// TwinCAT 3 PLC project Desktop
// ProgramVersion: 3.1.4020.1
// CompilerDefines: VISU_USEWSTRING
// libraries:
//   Standard, * (System)
//   VisuElems, 3.5.6.10 (System)
//   VisuElemsSpecialControls, 3.5.6.0 (System)
//   VisuElemsWinControls, 3.5.6.0 (System)
//   VisuElemTextEditor, 3.5.6.0 (System)
//   visuinputs, 3.5.6.0 (system)
//   VisuNativeControl, 3.5.6.0 (System)
//   Tc2_Math, * (Beckhoff Automation GmbH)
//   Tc2_MC2, * (Beckhoff Automation GmbH)
//   Tc2_NCI, * (Beckhoff Automation GmbH)
//   Tc2_NcKinematicTransformation, * (Beckhoff Automation GmbH)
//   Tc2_SPA, * (Beckhoff Automation GmbH)
//   Tc2_Standard, * (Beckhoff Automation GmbH)
//   Tc2_System, * (Beckhoff Automation GmbH)
//   Tc3_Interfaces, * (Beckhoff Automation GmbH)
//   Tc3_Module, * (Beckhoff Automation GmbH)
//   VisuDialogs, * (System)
// project tree:
//   / GlobalTextList.TcGTLO, PlcTask.TcTTO, Visualization Manager.TcVMO (not stored)
//   GVLs/ AxesCharacters.TcGVL, Functions.TcGVL, HardwareCharacters.TcGVL, ItpCharacters.TcGVL, KinCharacters.TcGVL
//   POUs/ Axes_Itp.TcPOU, Coordinate_System.TcPOU, Kinematics.TcPOU, Axes.TcPOU, Collision_Detection.TcPOU, MAIN.TcPOU, Home.TcPOU, Singularity.TcPOU, SoftFloat.TcPOU, UserFrames.TcPOU
//   VISUs/ CtrlPANEL.TcVIS, Home.TcVIS
// real-time tasks:
//   TASK PlcTask: cycle T#1ms, priority 1, ADS port 350
//   TASK VISU_TASK: cycle T#100000us, priority 10, ADS port 351
// motion (NC):
//   TASK NC-Task 1 SAF: cycle T#2ms, priority 4, ADS port 501
//   TASK NC-Task 1 SVB: cycle T#10ms, priority 8, ADS port 511
//   AXIS ACS M1 (id 1)
//     General: UnitName=Degree, UnitFlags=#x00000004
//     Dynamic: Acceleration=16333.3, Deceleration=16333.3, Jerk=111157
//     Velo: SlowManual=10, FastManual=20, Maximum=2500
//     OtherSettings: AllowMotionCmdToSlave=true
//     encoder EncType=1
//       EncPara: ScaleFactorNumerator=360, ScaleFactorDenominator=10485760, Offset=-437.0522
//         SoftEndMinControl: Enable=true, Range=-60
//         SoftEndMaxControl: Enable=true, Range=80
//     drive DrvType=5
//       Analog: VeloReferenz=2700
//       TimeComp: TaskDelayCycles=1
//     controller CtrType=1
//       CtrPara: PriorControlFactor=1
//         PID: PosKp=50
//         Observer: BandWidth=20
//   AXIS ACS M2 (id 2)
//     General: UnitName=Degree
//     Dynamic: Acceleration=16416.7, Deceleration=16416.7, Jerk=111137
//     Velo: SlowManual=10, FastManual=20, Maximum=2500
//     OtherSettings: AllowMotionCmdToSlave=true
//     encoder EncType=1
//       EncPara: ScaleFactorNumerator=360, ScaleFactorDenominator=10485760, Offset=-175.265
//         SoftEndMinControl: Enable=true, Range=-60
//         SoftEndMaxControl: Enable=true, Range=80
//     drive DrvType=5
//       Analog: VeloReferenz=2700
//       TimeComp: TaskDelayCycles=1
//     controller CtrType=1
//       CtrPara: PriorControlFactor=1
//         PID: PosKp=50
//         Observer: BandWidth=20
//   AXIS ACS M3 (id 3)
//     General: UnitName=Degree
//     Dynamic: Acceleration=16333.3, Deceleration=16333.3, Jerk=111157
//     Velo: SlowManual=10, FastManual=20, Maximum=2500
//     OtherSettings: AllowMotionCmdToSlave=true
//     encoder EncType=1
//       EncPara: ScaleFactorNumerator=360, ScaleFactorDenominator=10485760, Offset=-483.9976
//         SoftEndMinControl: Enable=true, Range=-60
//         SoftEndMaxControl: Enable=true, Range=80
//     drive DrvType=5
//       Analog: VeloReferenz=2700
//       TimeComp: TaskDelayCycles=1
//     controller CtrType=1
//       CtrPara: PriorControlFactor=1
//         PID: PosKp=50
//         Observer: BandWidth=20
//   AXIS MCS X (id 4)
//     Dynamic: Acceleration=16500, Deceleration=16500, Jerk=111122
//     Velo: SlowManual=50, FastManual=100, Maximum=2500
//     OtherSettings: AllowMotionCmdToSlave=true, PulseDistancePos=1, PulseDistanceNeg=1
//     encoder EncType=1
//       SoftEndMinControl: Range=-250
//       SoftEndMaxControl: Range=250
//     drive DrvType=5
//       Analog: VeloReferenz=3250
//       TimeComp: TaskDelayCycles=1
//     controller CtrType=1
//       CtrPara: PriorControlFactor=1
//         PID: PosKp=20
//         Observer: BandWidth=20
//   AXIS MCS Y (id 5)
//     Dynamic: Acceleration=16500, Deceleration=16500, Jerk=111122
//     Velo: SlowManual=50, FastManual=100, Maximum=2500
//     OtherSettings: AllowMotionCmdToSlave=true, PulseDistancePos=1, PulseDistanceNeg=1
//     encoder EncType=1
//       SoftEndMinControl: Range=-250
//       SoftEndMaxControl: Range=250
//     drive DrvType=5
//       Analog: VeloReferenz=3250
//       TimeComp: TaskDelayCycles=1
//     controller CtrType=1
//       CtrPara: PriorControlFactor=1
//         PID: PosKp=20
//         Observer: BandWidth=20
//   AXIS MCS Z (id 6)
//     Dynamic: Acceleration=16416.7, Deceleration=16416.7, Jerk=111137
//     Velo: SlowManual=50, FastManual=100, Maximum=2500
//     OtherSettings: AllowMotionCmdToSlave=true, PulseDistancePos=1, PulseDistanceNeg=1
//     encoder EncType=1
//       SoftEndMinControl: Range=-250
//       SoftEndMaxControl: Range=250
//     drive DrvType=5
//       Analog: VeloReferenz=3250
//       TimeComp: TaskDelayCycles=1
//     controller CtrType=1
//       CtrPara: PriorControlFactor=1
//         PID: PosKp=20
//         Observer: BandWidth=20
// variable links:
//   Desktop/Desktop Instance <-> NC-Task 1 SAF/Axes/ACS M1
//     PlcTask Inputs/AxesCharacters.MachX.NcToPlc <-> Outputs/ToPlc
//     PlcTask Outputs/AxesCharacters.MachX.PlcToNc <-> Inputs/FromPlc
//   Desktop/Desktop Instance <-> NC-Task 1 SAF/Axes/ACS M2
//     PlcTask Inputs/AxesCharacters.MachY.NcToPlc <-> Outputs/ToPlc
//     PlcTask Outputs/AxesCharacters.MachY.PlcToNc <-> Inputs/FromPlc
//   Desktop/Desktop Instance <-> NC-Task 1 SAF/Axes/ACS M3
//     PlcTask Inputs/AxesCharacters.MachZ.NcToPlc <-> Outputs/ToPlc
//     PlcTask Outputs/AxesCharacters.MachZ.PlcToNc <-> Inputs/FromPlc
//   Desktop/Desktop Instance <-> NC-Task 1 SAF/Axes/MCS X
//     PlcTask Inputs/AxesCharacters.SimsX.NcToPlc <-> Outputs/ToPlc
//     PlcTask Outputs/AxesCharacters.SimsX.PlcToNc <-> Inputs/FromPlc
//   Desktop/Desktop Instance <-> NC-Task 1 SAF/Axes/MCS Y
//     PlcTask Inputs/AxesCharacters.SimsY.NcToPlc <-> Outputs/ToPlc
//     PlcTask Outputs/AxesCharacters.SimsY.PlcToNc <-> Inputs/FromPlc
//   Desktop/Desktop Instance <-> NC-Task 1 SAF/Axes/MCS Z
//     PlcTask Inputs/AxesCharacters.SimsZ.NcToPlc <-> Outputs/ToPlc
//     PlcTask Outputs/AxesCharacters.SimsZ.PlcToNc <-> Inputs/FromPlc
//   Desktop/Desktop Instance <-> NC-Task 1 SAF/Kinametic_Channel
//     PlcTask Inputs/KinCharacters.in_stKinToPlc <-> Outputs/ToPlc
//     PlcTask Outputs/KinCharacters.out_stPlcTokin <-> Inputs/FromPlc
//   Desktop/Desktop Instance <-> NC-Task 1 SAF/NCI Interpolation
//     PlcTask Inputs/ItpCharacters.in_stItpToPLC <-> Outputs/ToPlc
//     PlcTask Outputs/ItpCharacters.out_stPLCToItp <-> Inputs/FromPlc

CONFIGURATION Desktop
    RESOURCE PLC ON TwinCAT3
        TASK PlcTask(INTERVAL := T#1ms, PRIORITY := 1);
        PROGRAM MAIN WITH PlcTask : MAIN;
    END_RESOURCE
END_CONFIGURATION

// ---- GVLs/AxesCharacters.TcGVL
VAR_GLOBAL
    in_uiMasterAxes_Override: LREAL := 100;
	in_bMasterAxes_Enable: BOOL ;    

    MachX: AXIS_REF;	
    in_bMachX_Enable: BOOL;
	in_uiMachX_Override: LREAL;
	out_bMachX_Status: BOOL;
	out_uiMachX_ErrorID: UDINT;
	
    MachY: AXIS_REF;
	in_bMachY_Enable: BOOL ;
	in_uiMachY_Override: LREAL;
	out_bMachY_Status: BOOL;
	out_uiMachY_ErrorID: UDINT;
	
    MachZ: AXIS_REF;
	in_bMachZ_Enable: BOOL ;
	in_uiMachZ_Override: LREAL;
	out_bMachZ_Status: BOOL;
	out_uiMachZ_ErrorID: UDINT;
	
    SimsX: AXIS_REF;
	in_bSimsX_Enable: BOOL ;
	in_uiSimsX_Override: LREAL;
	out_bSimsX_Status: BOOL;
	out_uiSimsX_ErrorID: UDINT;
	
    SimsY: AXIS_REF;
	in_bSimsY_Enable: BOOL ;
	in_uiSimsY_Override: LREAL;
	out_bSimsY_Status: BOOL;
	out_uiSimsY_ErrorID: UDINT;
	
    SimsZ: AXIS_REF;
	in_bSimsZ_Enable: BOOL ;
	in_uiSimsZ_Override: LREAL;
	out_bSimsZ_Status: BOOL;
	out_uiSimsZ_ErrorID: UDINT;
		
	in_bAxes_MachX_Jog_Forward: BOOL;
	in_bAxes_MachX_Jog_Backward: BOOL;
	out_uiAxes_MachX_Jog_ErrorID: UDINT;
		
	in_bAxes_MachY_Jog_Forward: BOOL;
	in_bAxes_MachY_Jog_Backward: BOOL;
	out_uiAxes_MachY_Jog_ErrorID: UDINT;
	
	in_bAxes_MachZ_Jog_Forward: BOOL;
	in_bAxes_MachZ_Jog_Backward: BOOL;
	out_uiAxes_MachZ_Jog_ErrorID: UDINT;
	
    in_bAxes_SimsX_Jog_Forward: BOOL;
	in_bAxes_SimsX_Jog_Backward: BOOL;
	out_uiAxes_SimsX_Jog_ErrorID: UDINT;
	
    in_bAxes_SimsY_Jog_Forward: BOOL;
	in_bAxes_SimsY_Jog_Backward: BOOL;
	out_uiAxes_SimsY_Jog_ErrorID: UDINT;
	
    in_bAxes_SimsZ_Jog_Forward: BOOL;
	in_bAxes_SimsZ_Jog_Backward: BOOL;
	out_uiAxes_SimsZ_Jog_ErrorID: UDINT;

	out_uiMachX_Error: BOOL;
	out_uiMachY_Error: BOOL;
	out_uiMachZ_Error: BOOL;
	out_uiSimsX_Error: BOOL;
	out_uiSimsY_Error: BOOL;
	out_uiSimsZ_Error: BOOL;
	out_bAxes_Master_Error: BOOL;
	
	Axes_Reset_All: BOOL;
		
END_VAR

// ---- GVLs/Functions.TcGVL
VAR_GLOBAL
	
// Move to Home Function
	in_b_MoveHome: BOOL;
	SimsX_Home_Done: BOOL;
	SimsY_Home_Done: BOOL;
	SimsZ_Home_Done: BOOL;
	
	Set_Pos_XHome: LREAL;
	Set_Pos_YHome: LREAL;
	Set_Pos_ZHome: LREAL;
	Set_Home_Override: LREAL:= 1000;
	out_b_inHome: BOOL;
	
END_VAR

// ---- GVLs/HardwareCharacters.TcGVL
VAR_GLOBAL
	in_bMasterAxes_Enable_HW AT %I*: BOOL;
	out_bMasterAxes_Enable_HW AT %Q*: BOOL;
	out_bSimsX_Axes_busy_HW AT %Q*: BOOL;
	out_bSimsY_Axes_busy_HW AT %Q*: BOOL;
	out_bSimsZ_Axes_busy_HW AT %Q*: BOOL;
	in_bAxes_SimsX_Jog_Forward_HW AT %I*: BOOL;
	in_bAxes_SimsX_Jog_Backward_HW AT %I*: BOOL;
	in_bAxes_SimsY_Jog_Forward_HW AT %I*: BOOL;
	in_bAxes_SimsY_Jog_Backward_HW AT %I*: BOOL;
	in_bAxes_SimsZ_Jog_Forward_HW AT %I*: BOOL;
	in_bAxes_SimsZ_Jog_Backward_HW AT %I*: BOOL;
	in_bTOOL_HW AT %I*: BOOL;
	out_bTOOL_HW AT %Q*: BOOL;
	in_uiMasterAxes_Override_HW1 AT %I*: BOOL;
	in_uiMasterAxes_Override_HW2 AT %I*: BOOL;
	iXTrq_feedback AT %I*:INT;
END_VAR

// ---- GVLs/ItpCharacters.TcGVL
VAR_GLOBAL
	
    in_bAxes_ItpLoadPRG_Execute: BOOL;
	in_strAxes_ItpLoadPRG_PRGPath: STRING :='Pick_place.nc';
	in_bAxes_ItpLoadPRG_Busy: BOOL;
	out_uiAxes_ItpLoadPRG_ErrorID: UDINT;
	
    in_bAxes_ItpStartStop_Error: BOOL;
	in_bAxes_ItpStartStop_Start: BOOL;
	in_bAxes_ItpStartStop_Stop: BOOL;
	in_bAxes_ItpStartStop_Busy: BOOL;
	in_uiAxes_ItpStartStop_ErrorID: UDINT;
	
    in_bAxes_BuildItpGoup_Execute: BOOL;
	out_bAxes_BuildItpGoup_Busy: BOOL;
	out_uiAxes_BuildItpGoup_ErrorID: UDINT;
	out_bAxes_BuildItpGoup_Error: BOOL;
	out_bAxes_ItpLoadPRG_Error: BOOL;
	
    in_bAxes_ItpReset_Group_Execute: BOOL;
	out_bAxes_ItpReset_Group_Error: BOOL;
	out_uiAxes_ItpReset_Group_ErrorID: UDINT;
	
    in_stItpToPLC AT %I*: NCTOPLC_NCICHANNEL_REF;
	out_stPLCToItp AT %Q*: PLCTONC_NCICHANNEL_REF;
	
	out_uiItp_InterpreterState AT %I*: UINT;
	out_wdItp_InterpolationMode AT %I*: WORD;
	out_uiItp_Linenumber AT %I*: UDINT;
	out_uiItp_Mcodenumber AT %I*: UINT;
	out_uiItp_ErrorEncountered AT %I*: UDINT;
	out_uiItp_Feedrate AT %I*: LREAL;

	out_bAxes_BuildItpGoup_Done: BOOL;
	out_bAxes_ItpReset_Group_Busy: BOOL;
	out_stItp_InterpreterState_String: WSTRING(255);
	out_bAxes_ItpLoadPRG_DoneHMI: BOOL;
	out_wdItp_InterpolationMode_string: WSTRING;
	in_bAxes_ItpReConfig_Group_Execute: BOOL;
	in_bAxes_ItpReConfig_Group_Busy: BOOL;
	in_bAxes_ItpReConfig_Group_Busy_HMI: BOOL;
	
	in_bAxes_ItpConfirmHSK_Execute: BOOL;
	out_bAxes_ItpConfirmHSK_Busy: BOOL;
	in_bTOOL: BOOL;

END_VAR

// ---- GVLs/KinCharacters.TcGVL
VAR_GLOBAL
	in_bAxes_KinConfigGroup_Execute: BOOL;
	out_bAxes_KinConfigGroup_Done: BOOL;
    out_uiAxes_KinConfigGroup_ErrorID: UDINT;
	
    in_bAxes_KinResetGroup_Execute: BOOL;
	out_bAxes_KinResetGroup_Done: BOOL;
	out_uiAxes_KinResetGroup_ErrorID: UDINT;
	
	st_Axes_Kin: ST_KinAxes;
	
	in_stKinToPlc AT %I*: NCTOPLC_NCICHANNEL_REF;
	out_stPlcTokin AT %Q*: PLCTONC_NCICHANNEL_REF;
    out_bAxes_KinConfigGroup_Error: BOOL;
	out_bAxes_KinResetGroup_Error: BOOL;
	
	out_bAxes_KinConfigGroup_Done_HMI: BOOL;
END_VAR

// ---- POUs/MAIN.TcPOU
PROGRAM MAIN
VAR

END_VAR

Axes();
Kinematics();
Home();
Singularity();

END_PROGRAM

// ---- POUs/Axes.TcPOU
PROGRAM Axes
VAR
	Fb_MachX_Power: MC_Power;
	Fb_MachY_Power: MC_Power;
	Fb_MachZ_Power: MC_Power;
	Fb_SimsX_Power: MC_Power;
	Fb_SimsY_Power: MC_Power;
	Fb_SimsZ_Power: MC_Power;

	Fb_Axes_MachX_Reset: MC_Reset;
	Fb_Axes_MachY_Reset: MC_Reset;
	Fb_Axes_MachZ_Reset: MC_Reset;
	Fb_Axes_SimsX_Reset: MC_Reset;
	Fb_Axes_SimsY_Reset: MC_Reset;
	Fb_Axes_SimsZ_Reset: MC_Reset;
	
	fb_Axes_MachX_Jog: MC_Jog;
	fb_Axes_MachY_Jog: MC_Jog;
	fb_Axes_MachZ_Jog: MC_Jog;
	fb_Axes_SimsX_Jog: MC_Jog;
	fb_Axes_SimsY_Jog: MC_Jog;
	fb_Axes_SimsZ_Jog: MC_Jog;
	bo_override: BOOL;
	bo_tp_override: TP;
END_VAR

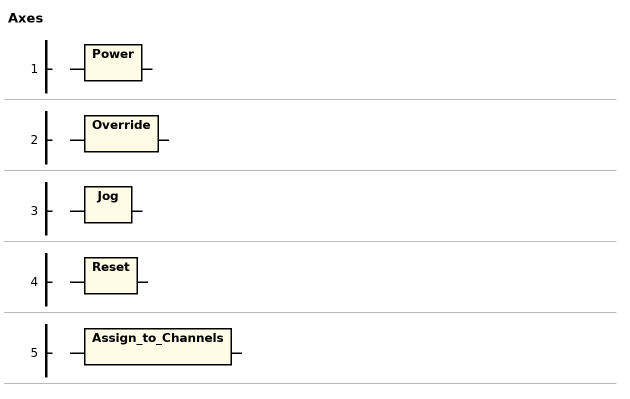
// NETWORK 1
Power();

// NETWORK 2
Override();

// NETWORK 3
Jog();

// NETWORK 4
Reset();

// NETWORK 5
Assign_to_Channels();

ACTION Assign_to_Channels:
st_Axes_Kin.nAxisIdsAcs[1]	:= MachX.NcToPlc.AxisId;
st_Axes_Kin.nAxisIdsAcs[2]	:= MachY.NcToPlc.AxisId;
st_Axes_Kin.nAxisIdsAcs[3]	:= MachZ.NcToPlc.AxisId;
st_Axes_Kin.nAxisIdsMcs[1]	:= SimsX.NcToPlc.AxisId;
st_Axes_Kin.nAxisIdsMcs[2]	:= SimsY.NcToPlc.AxisId;
st_Axes_Kin.nAxisIdsMcs[3]	:= SimsZ.NcToPlc.AxisId;
END_ACTION

ACTION Jog:
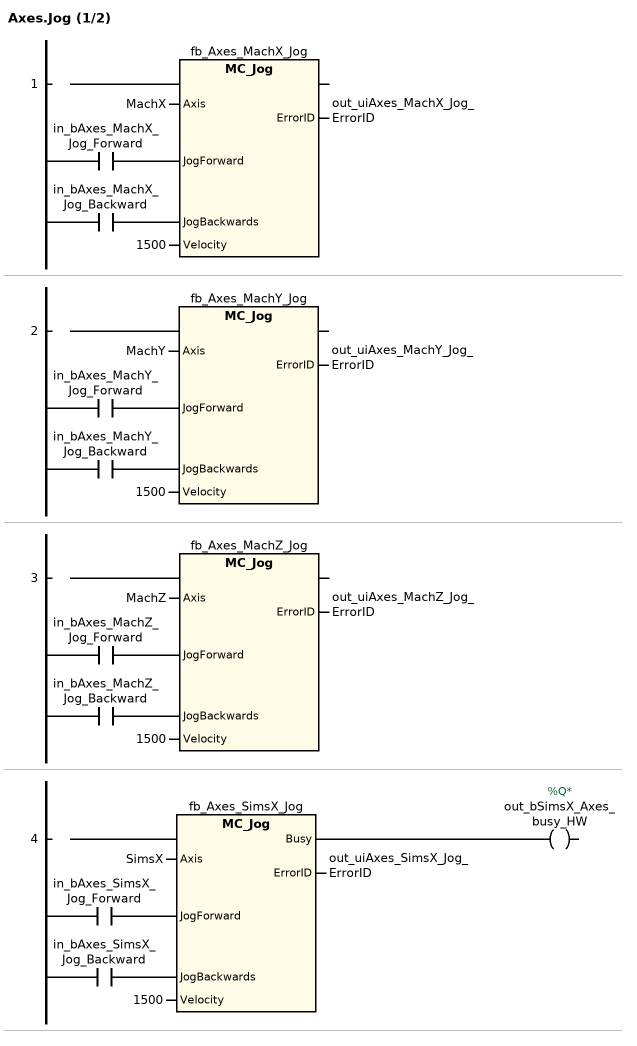
// NETWORK 1
fb_Axes_MachX_Jog(
    Axis := MachX,
    JogForward := in_bAxes_MachX_Jog_Forward,
    JogBackwards := in_bAxes_MachX_Jog_Backward,
    Velocity := 1500,
    ErrorID => out_uiAxes_MachX_Jog_ErrorID); // MC_Jog

// NETWORK 2
fb_Axes_MachY_Jog(
    Axis := MachY,
    JogForward := in_bAxes_MachY_Jog_Forward,
    JogBackwards := in_bAxes_MachY_Jog_Backward,
    Velocity := 1500,
    ErrorID => out_uiAxes_MachY_Jog_ErrorID); // MC_Jog

// NETWORK 3
fb_Axes_MachZ_Jog(
    Axis := MachZ,
    JogForward := in_bAxes_MachZ_Jog_Forward,
    JogBackwards := in_bAxes_MachZ_Jog_Backward,
    Velocity := 1500,
    ErrorID => out_uiAxes_MachZ_Jog_ErrorID); // MC_Jog

// NETWORK 4
//   out_bSimsX_Axes_busy_HW: AT %Q*
fb_Axes_SimsX_Jog(
    Axis := SimsX,
    JogForward := in_bAxes_SimsX_Jog_Forward,
    JogBackwards := in_bAxes_SimsX_Jog_Backward,
    Velocity := 1500,
    ErrorID => out_uiAxes_SimsX_Jog_ErrorID); // MC_Jog
out_bSimsX_Axes_busy_HW := fb_Axes_SimsX_Jog.Busy;

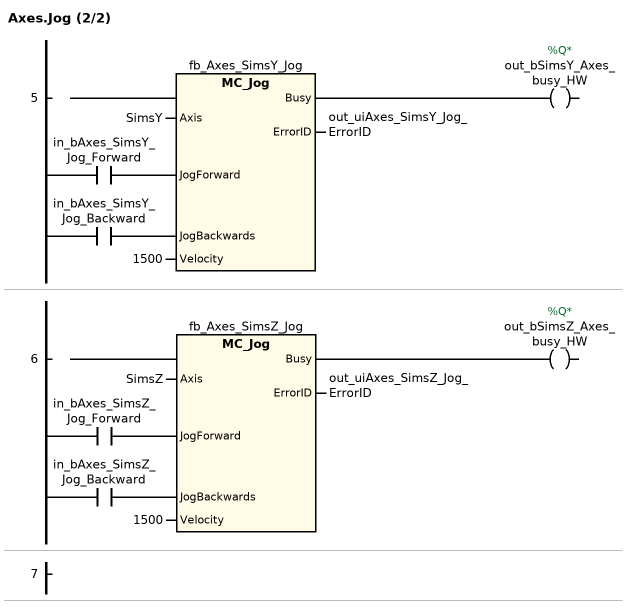
// NETWORK 5
//   out_bSimsY_Axes_busy_HW: AT %Q*
fb_Axes_SimsY_Jog(
    Axis := SimsY,
    JogForward := in_bAxes_SimsY_Jog_Forward,
    JogBackwards := in_bAxes_SimsY_Jog_Backward,
    Velocity := 1500,
    ErrorID => out_uiAxes_SimsY_Jog_ErrorID); // MC_Jog
out_bSimsY_Axes_busy_HW := fb_Axes_SimsY_Jog.Busy;

// NETWORK 6
//   out_bSimsZ_Axes_busy_HW: AT %Q*
fb_Axes_SimsZ_Jog(
    Axis := SimsZ,
    JogForward := in_bAxes_SimsZ_Jog_Forward,
    JogBackwards := in_bAxes_SimsZ_Jog_Backward,
    Velocity := 1500,
    ErrorID => out_uiAxes_SimsZ_Jog_ErrorID); // MC_Jog
out_bSimsZ_Axes_busy_HW := fb_Axes_SimsZ_Jog.Busy;

// NETWORK 7
END_ACTION

ACTION Override:
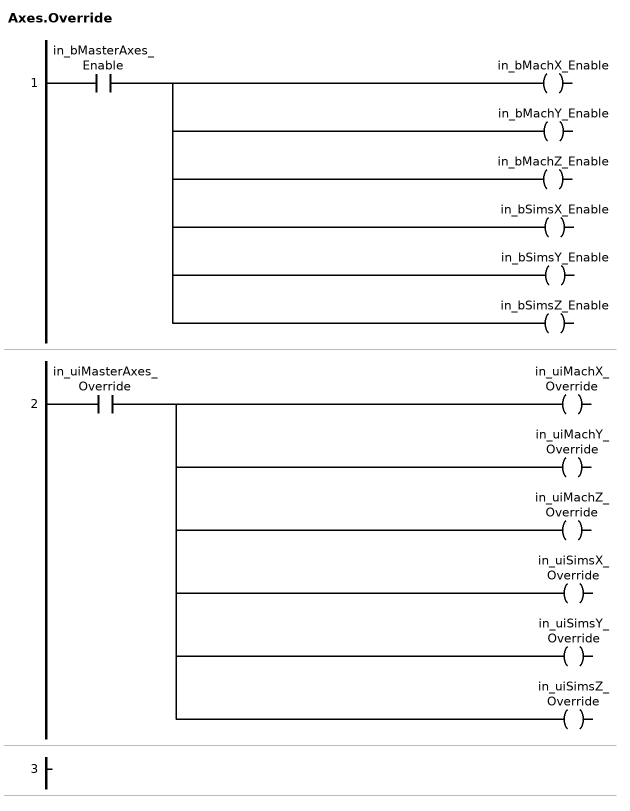
// NETWORK 1
in_bMachX_Enable := in_bMasterAxes_Enable;
in_bMachY_Enable := in_bMasterAxes_Enable;
in_bMachZ_Enable := in_bMasterAxes_Enable;
in_bSimsX_Enable := in_bMasterAxes_Enable;
in_bSimsY_Enable := in_bMasterAxes_Enable;
in_bSimsZ_Enable := in_bMasterAxes_Enable;

// NETWORK 2
in_uiMachX_Override := in_uiMasterAxes_Override;
in_uiMachY_Override := in_uiMasterAxes_Override;
in_uiMachZ_Override := in_uiMasterAxes_Override;
in_uiSimsX_Override := in_uiMasterAxes_Override;
in_uiSimsY_Override := in_uiMasterAxes_Override;
in_uiSimsZ_Override := in_uiMasterAxes_Override;

// NETWORK 3
END_ACTION

ACTION Power:
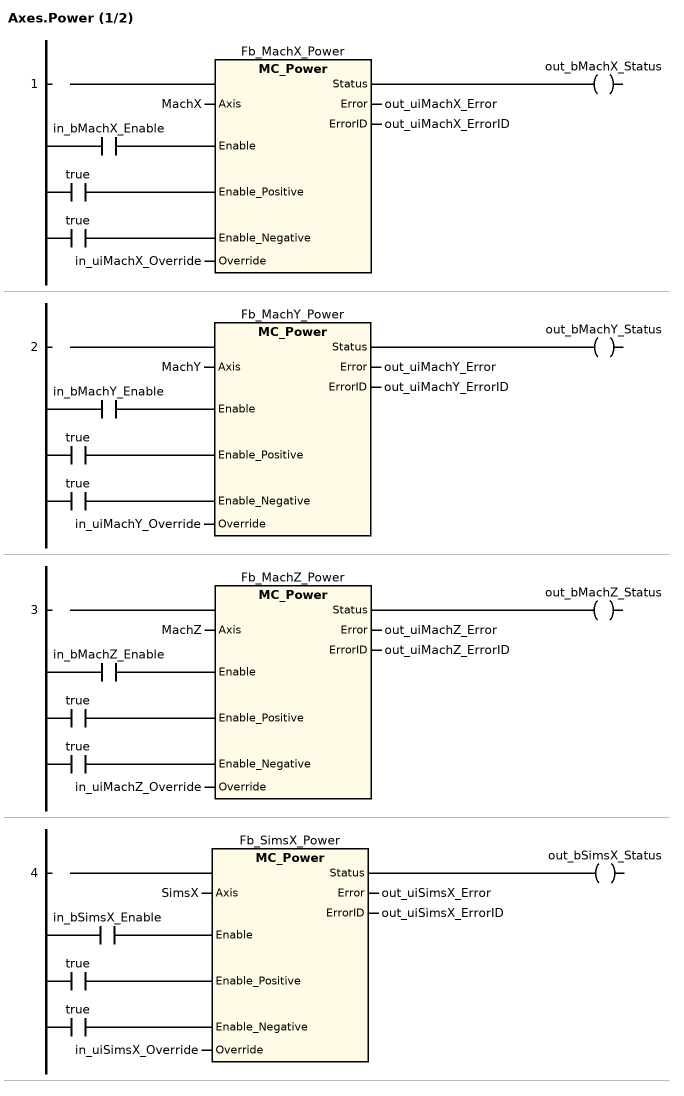
// NETWORK 1
Fb_MachX_Power(
    Axis := MachX,
    Enable := in_bMachX_Enable,
    Enable_Positive := true,
    Enable_Negative := true,
    Override := in_uiMachX_Override,
    Error => out_uiMachX_Error,
    ErrorID => out_uiMachX_ErrorID); // MC_Power
out_bMachX_Status := Fb_MachX_Power.Status;

// NETWORK 2
Fb_MachY_Power(
    Axis := MachY,
    Enable := in_bMachY_Enable,
    Enable_Positive := true,
    Enable_Negative := true,
    Override := in_uiMachY_Override,
    Error => out_uiMachY_Error,
    ErrorID => out_uiMachY_ErrorID); // MC_Power
out_bMachY_Status := Fb_MachY_Power.Status;

// NETWORK 3
Fb_MachZ_Power(
    Axis := MachZ,
    Enable := in_bMachZ_Enable,
    Enable_Positive := true,
    Enable_Negative := true,
    Override := in_uiMachZ_Override,
    Error => out_uiMachZ_Error,
    ErrorID => out_uiMachZ_ErrorID); // MC_Power
out_bMachZ_Status := Fb_MachZ_Power.Status;

// NETWORK 4
Fb_SimsX_Power(
    Axis := SimsX,
    Enable := in_bSimsX_Enable,
    Enable_Positive := true,
    Enable_Negative := true,
    Override := in_uiSimsX_Override,
    Error => out_uiSimsX_Error,
    ErrorID => out_uiSimsX_ErrorID); // MC_Power
out_bSimsX_Status := Fb_SimsX_Power.Status;

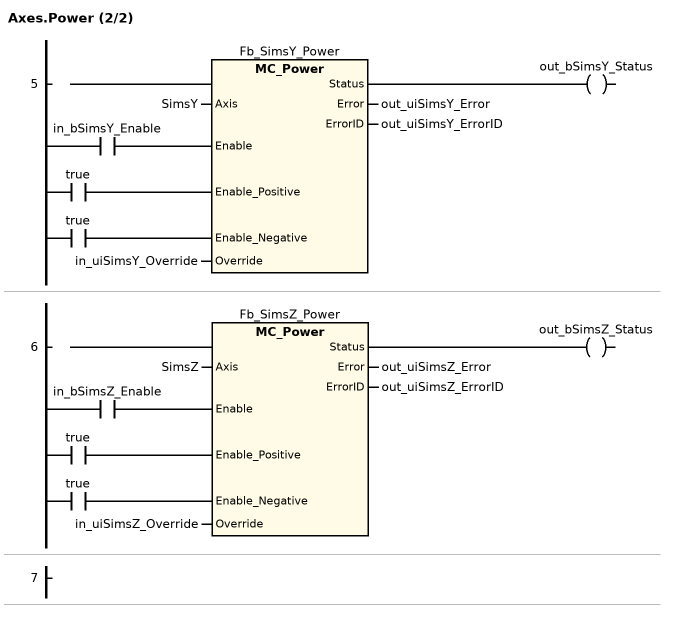
// NETWORK 5
Fb_SimsY_Power(
    Axis := SimsY,
    Enable := in_bSimsY_Enable,
    Enable_Positive := true,
    Enable_Negative := true,
    Override := in_uiSimsY_Override,
    Error => out_uiSimsY_Error,
    ErrorID => out_uiSimsY_ErrorID); // MC_Power
out_bSimsY_Status := Fb_SimsY_Power.Status;

// NETWORK 6
Fb_SimsZ_Power(
    Axis := SimsZ,
    Enable := in_bSimsZ_Enable,
    Enable_Positive := true,
    Enable_Negative := true,
    Override := in_uiSimsZ_Override,
    Error => out_uiSimsZ_Error,
    ErrorID => out_uiSimsZ_ErrorID); // MC_Power
out_bSimsZ_Status := Fb_SimsZ_Power.Status;

// NETWORK 7
END_ACTION

ACTION Reset:
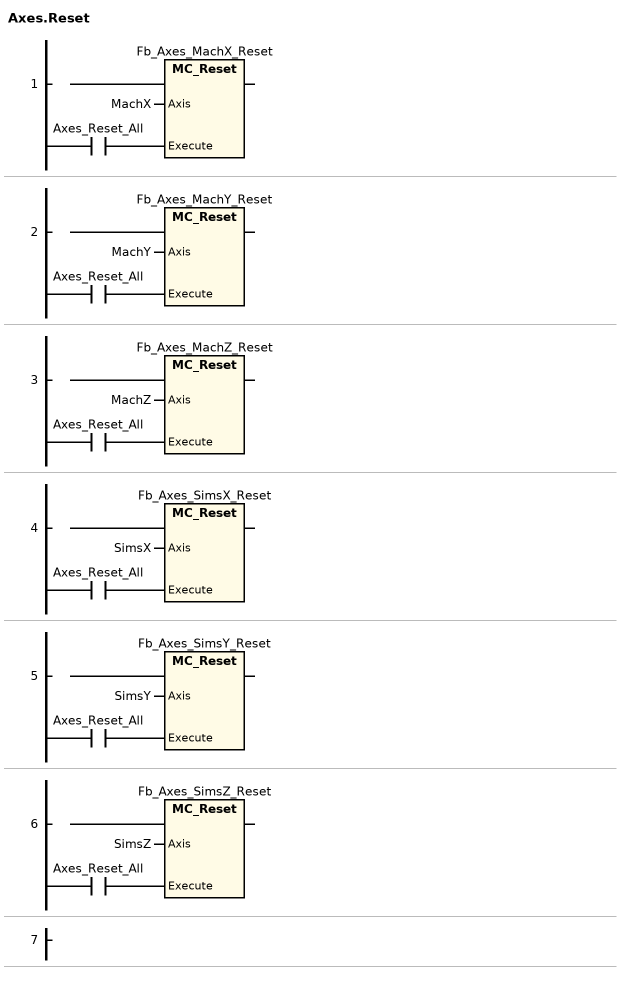
// NETWORK 1
Fb_Axes_MachX_Reset(Axis := MachX, Execute := Axes_Reset_All); // MC_Reset

// NETWORK 2
Fb_Axes_MachY_Reset(Axis := MachY, Execute := Axes_Reset_All); // MC_Reset

// NETWORK 3
Fb_Axes_MachZ_Reset(Axis := MachZ, Execute := Axes_Reset_All); // MC_Reset

// NETWORK 4
Fb_Axes_SimsX_Reset(Axis := SimsX, Execute := Axes_Reset_All); // MC_Reset

// NETWORK 5
Fb_Axes_SimsY_Reset(Axis := SimsY, Execute := Axes_Reset_All); // MC_Reset

// NETWORK 6
Fb_Axes_SimsZ_Reset(Axis := SimsZ, Execute := Axes_Reset_All); // MC_Reset

// NETWORK 7
END_ACTION

END_PROGRAM

// ---- POUs/Kinematics.TcPOU
PROGRAM Kinematics
VAR
	Fb_Axes_KinCongifGroup: FB_KinConfigGroup;
	Fb_Axes_KinResetGroup: FB_KinResetGroup;
	Fb_Axes_KinReConfigGroup: CfgReconfigGroup;
	Build_Kin_Group: TOF;
	Trig_Build: BOOL;
	bb_tp_reset: BOOL;
	BB_TP_Kin: TP;
END_VAR

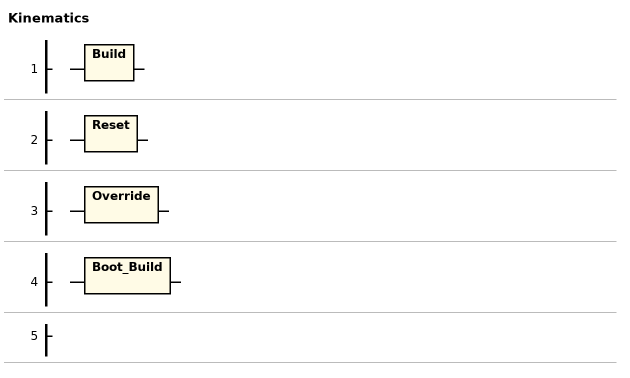
// NETWORK 1
Build();

// NETWORK 2
Reset();

// NETWORK 3
Override();

// NETWORK 4
Boot_Build();

// NETWORK 5

ACTION Boot_Build:
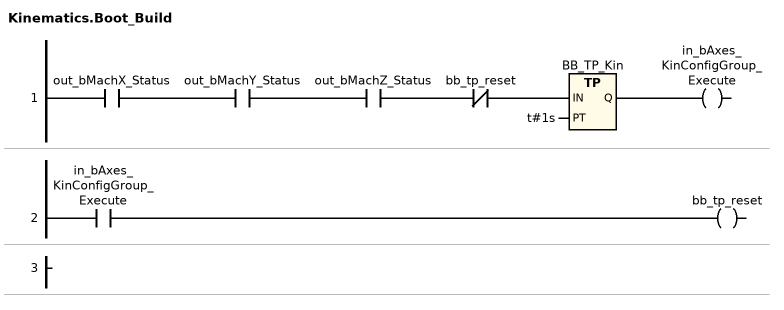
// NETWORK 1
BB_TP_Kin(IN := out_bMachX_Status AND out_bMachY_Status AND out_bMachZ_Status AND NOT bb_tp_reset, PT := t#1s); // TP
in_bAxes_KinConfigGroup_Execute := BB_TP_Kin.Q;

// NETWORK 2
bb_tp_reset := in_bAxes_KinConfigGroup_Execute;

// NETWORK 3
END_ACTION

ACTION Build:
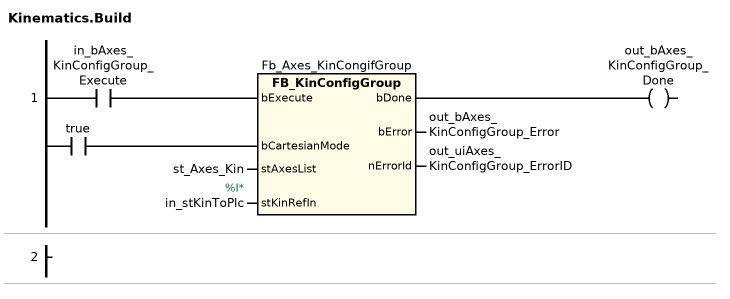
// NETWORK 1
//   in_stKinToPlc: AT %I*
Fb_Axes_KinCongifGroup(
    bExecute := in_bAxes_KinConfigGroup_Execute,
    bCartesianMode := true,
    stAxesList := st_Axes_Kin,
    stKinRefIn := in_stKinToPlc,
    bError => out_bAxes_KinConfigGroup_Error,
    nErrorId => out_uiAxes_KinConfigGroup_ErrorID); // FB_KinConfigGroup
out_bAxes_KinConfigGroup_Done := Fb_Axes_KinCongifGroup.bDone;

// NETWORK 2
END_ACTION

ACTION Override:
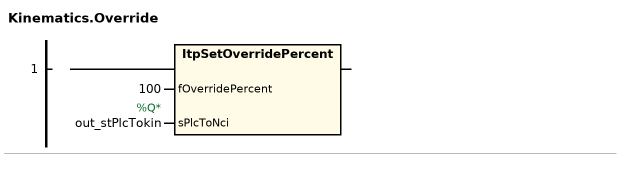
// NETWORK 1
//   out_stPlcTokin: AT %Q*
ItpSetOverridePercent(fOverridePercent := 100, sPlcToNci := out_stPlcTokin);
END_ACTION

ACTION Reset:
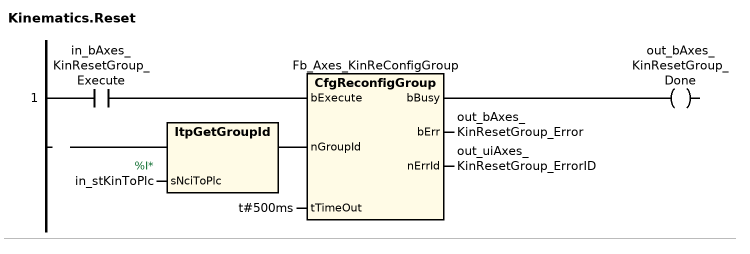
// NETWORK 1
//   in_stKinToPlc: AT %I*
Fb_Axes_KinReConfigGroup(
    bExecute := in_bAxes_KinResetGroup_Execute,
    nGroupId := ItpGetGroupId(sNciToPlc := in_stKinToPlc),
    tTimeOut := t#500ms,
    bErr => out_bAxes_KinResetGroup_Error,
    nErrId => out_uiAxes_KinResetGroup_ErrorID); // CfgReconfigGroup
out_bAxes_KinResetGroup_Done := Fb_Axes_KinReConfigGroup.bBusy;
END_ACTION

END_PROGRAM

// ---- POUs/Home.TcPOU
PROGRAM Home
VAR
	SimsX_Home: MC_MoveAbsolute;
	SimsX_Home_ErrorID: UDINT;
	SimsY_Home: MC_MoveAbsolute;
	SimsZ_Home: MC_MoveAbsolute;
	SimsY_Home_ErrorID: UDINT;
	SimsZ_Home_ErrorID: UDINT;
	Inside_Dia: LREAL;
	Pos_Exists: BOOL;
	Pos_NotValid: BOOL;
END_VAR

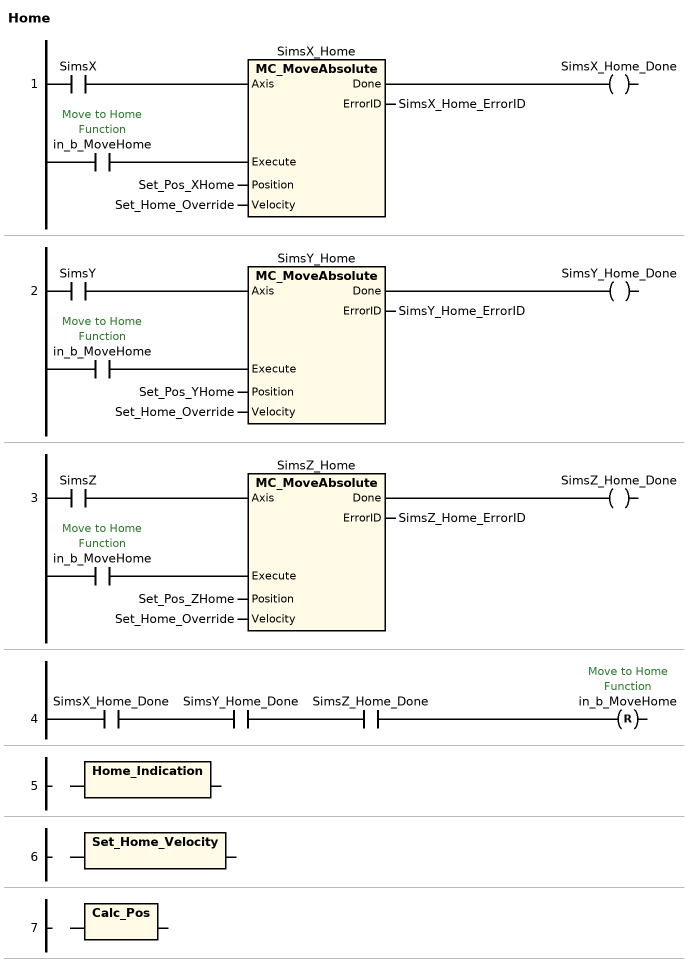
// NETWORK 1
//   in_b_MoveHome: Move to Home Function
SimsX_Home(
    Axis := SimsX,
    Execute := in_b_MoveHome,
    Position := Set_Pos_XHome,
    Velocity := Set_Home_Override,
    ErrorID => SimsX_Home_ErrorID); // MC_MoveAbsolute
SimsX_Home_Done := SimsX_Home.Done;

// NETWORK 2
//   in_b_MoveHome: Move to Home Function
SimsY_Home(
    Axis := SimsY,
    Execute := in_b_MoveHome,
    Position := Set_Pos_YHome,
    Velocity := Set_Home_Override,
    ErrorID => SimsY_Home_ErrorID); // MC_MoveAbsolute
SimsY_Home_Done := SimsY_Home.Done;

// NETWORK 3
//   in_b_MoveHome: Move to Home Function
SimsZ_Home(
    Axis := SimsZ,
    Execute := in_b_MoveHome,
    Position := Set_Pos_ZHome,
    Velocity := Set_Home_Override,
    ErrorID => SimsZ_Home_ErrorID); // MC_MoveAbsolute
SimsZ_Home_Done := SimsZ_Home.Done;

// NETWORK 4
//   in_b_MoveHome: Move to Home Function
in_b_MoveHome R= SimsX_Home_Done AND SimsY_Home_Done AND SimsZ_Home_Done;

// NETWORK 5
Home_Indication();

// NETWORK 6
Set_Home_Velocity();

// NETWORK 7
Calc_Pos();

ACTION Calc_Pos:
Inside_Dia:= SQRT((Set_Pos_XHome)*(Set_Pos_XHome)+
				  (Set_Pos_YHome)*(Set_Pos_YHome));
				  
IF Inside_Dia>=251 OR Set_Pos_ZHome>=70 OR Set_Pos_ZHome<=-160 THEN
	Pos_Exists:=FALSE;	
	Pos_NotValid:=TRUE;
ELSE
	Pos_Exists:=TRUE;
	Pos_NotValid:=FALSE;
END_IF
END_ACTION

ACTION Home_Indication:
IF (Set_Pos_XHome <= (SimsX.NcToPlc.ActPos+0.5) AND  Set_Pos_XHome >= (SimsX.NcToPlc.ActPos-0.5)) AND
   (Set_Pos_YHome <= (SimsY.NcToPlc.ActPos+0.5) AND  Set_Pos_YHome >= (SimsY.NcToPlc.ActPos-0.5)) AND
   (Set_Pos_ZHome <= (SimsZ.NcToPlc.ActPos+0.5) AND  Set_Pos_ZHome >= (SimsZ.NcToPlc.ActPos-0.5))
 THEN
	out_b_inHome := TRUE;
ELSE
	out_b_inHome := FALSE;
END_IF
END_ACTION

ACTION Set_Home_Velocity:

Set_Home_Override := (Set_Home_Override*(in_uiMasterAxes_Override/100));
END_ACTION

END_PROGRAM

// ---- POUs/Singularity.TcPOU
PROGRAM Singularity
VAR
	Inside_Dia: LREAL;
	At_Singularity: BOOL;
	Near_Singularity: BOOL;
	Singular_SimsX_Stop: MC_Stop;
	Singular_SimsY_Stop: MC_Stop;
	Singular_SimsZ_Stop: MC_Stop;
END_VAR

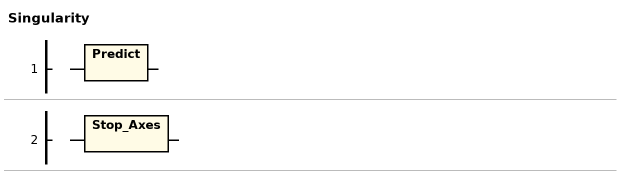
// NETWORK 1
Predict();

// NETWORK 2
Stop_Axes();

ACTION Predict:
Inside_Dia:= SQRT((SimsX.NcToPlc.ActPos)*(SimsX.NcToPlc.ActPos)+
				  (SimsY.NcToPlc.ActPos)*(SimsY.NcToPlc.ActPos));
		
IF Inside_Dia>=249 OR SimsZ.NcToPlc.ActPos>=65 OR SimsZ.NcToPlc.ActPos<=-155 THEN
	At_Singularity:=TRUE;
ELSE
	At_Singularity:=FALSE;	
END_IF

IF Inside_Dia>=240 OR SimsZ.NcToPlc.ActPos>=60 OR SimsZ.NcToPlc.ActPos<=-150 THEN
	Near_Singularity:=TRUE;
ELSE
	Near_Singularity:=FALSE;	
END_IF
END_ACTION

ACTION Reset:
// NETWORK 1
END_ACTION

ACTION Stop_Axes:
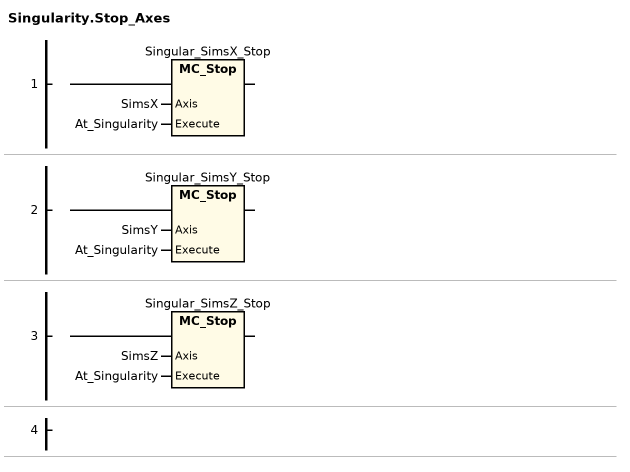
// NETWORK 1
Singular_SimsX_Stop(Axis := SimsX, Execute := At_Singularity); // MC_Stop

// NETWORK 2
Singular_SimsY_Stop(Axis := SimsY, Execute := At_Singularity); // MC_Stop

// NETWORK 3
Singular_SimsZ_Stop(Axis := SimsZ, Execute := At_Singularity); // MC_Stop

// NETWORK 4
END_ACTION

END_PROGRAM

// ---- POUs/Axes_Itp.TcPOU
PROGRAM Axes_Itp
VAR
	Fb_Axes_ItpLoadProg: ItpLoadProg;
	Fb_Axes_ItpStartStop: ItpStartStop;
	Fb_Axes_BuildItpGoup: CfgBuild3DGroup;
    localstr: STRING;
	localconstr: STRING(255);
	Fb_Axes_ItpReset_Group: ItpReset;
	
	Fb_Axes_ItpReConfig_Group: CfgReconfigGroup;
	Fb_Axes_ItpConfirmHSK: ItpConfirmHsk;
	
	M_code_rtrig: R_TRIG;
	bItpGet_MHsk: bool;
	nItp_MhskNumber: INT;
	nstep: INT;
END_VAR

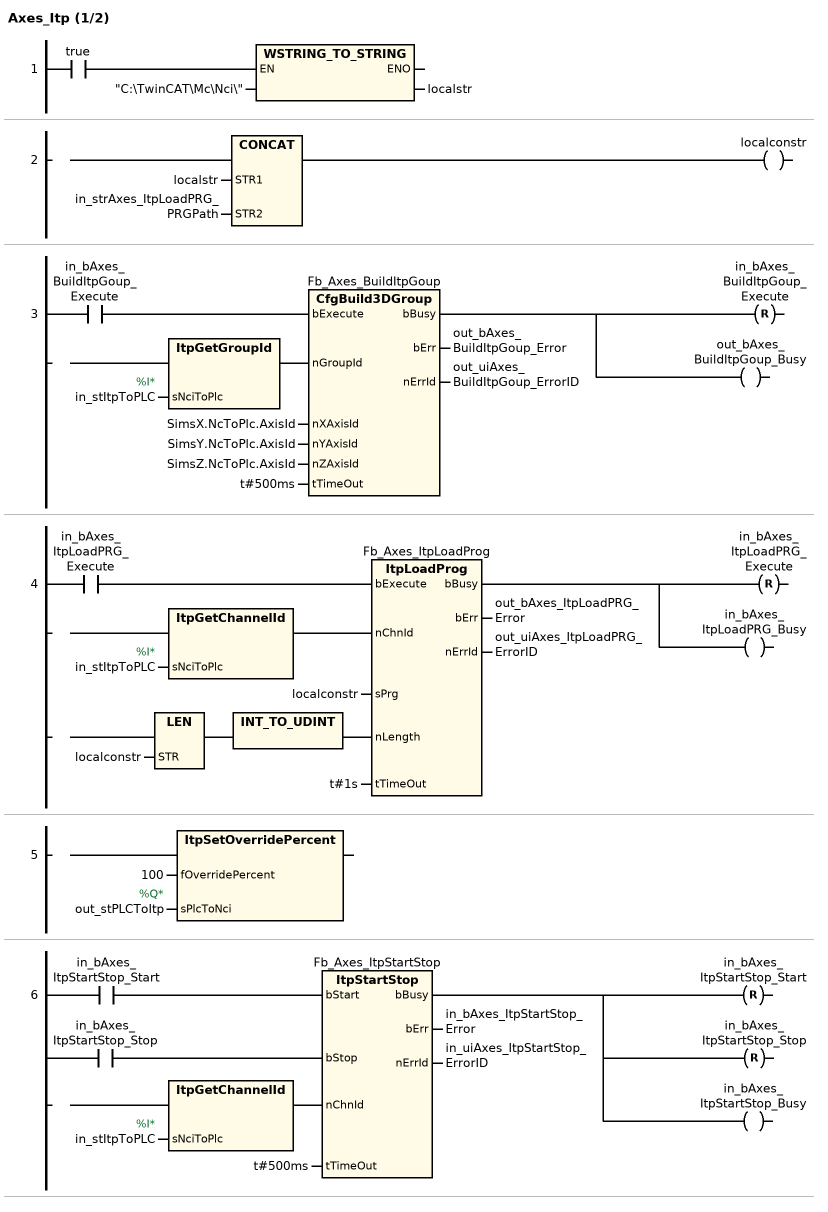
// NETWORK 1
IF true THEN localstr := WSTRING_TO_STRING("C:\TwinCAT\Mc\Nci\"); END_IF

// NETWORK 2
localconstr := CONCAT(STR1 := localstr, STR2 := in_strAxes_ItpLoadPRG_PRGPath);

// NETWORK 3
//   in_stItpToPLC: AT %I*
Fb_Axes_BuildItpGoup(
    bExecute := in_bAxes_BuildItpGoup_Execute,
    nGroupId := ItpGetGroupId(sNciToPlc := in_stItpToPLC),
    nXAxisId := SimsX.NcToPlc.AxisId,
    nYAxisId := SimsY.NcToPlc.AxisId,
    nZAxisId := SimsZ.NcToPlc.AxisId,
    tTimeOut := t#500ms,
    bErr => out_bAxes_BuildItpGoup_Error,
    nErrId => out_uiAxes_BuildItpGoup_ErrorID); // CfgBuild3DGroup
in_bAxes_BuildItpGoup_Execute R= Fb_Axes_BuildItpGoup.bBusy;
out_bAxes_BuildItpGoup_Busy := Fb_Axes_BuildItpGoup.bBusy;

// NETWORK 4
//   in_stItpToPLC: AT %I*
Fb_Axes_ItpLoadProg(
    bExecute := in_bAxes_ItpLoadPRG_Execute,
    nChnId := ItpGetChannelId(sNciToPlc := in_stItpToPLC),
    sPrg := localconstr,
    nLength := INT_TO_UDINT(LEN(STR := localconstr)),
    tTimeOut := t#1s,
    bErr => out_bAxes_ItpLoadPRG_Error,
    nErrId => out_uiAxes_ItpLoadPRG_ErrorID); // ItpLoadProg
in_bAxes_ItpLoadPRG_Execute R= Fb_Axes_ItpLoadProg.bBusy;
in_bAxes_ItpLoadPRG_Busy := Fb_Axes_ItpLoadProg.bBusy;

// NETWORK 5
//   out_stPLCToItp: AT %Q*
ItpSetOverridePercent(fOverridePercent := 100, sPlcToNci := out_stPLCToItp);

// NETWORK 6
//   in_stItpToPLC: AT %I*
Fb_Axes_ItpStartStop(
    bStart := in_bAxes_ItpStartStop_Start,
    bStop := in_bAxes_ItpStartStop_Stop,
    nChnId := ItpGetChannelId(sNciToPlc := in_stItpToPLC),
    tTimeOut := t#500ms,
    bErr => in_bAxes_ItpStartStop_Error,
    nErrId => in_uiAxes_ItpStartStop_ErrorID); // ItpStartStop
in_bAxes_ItpStartStop_Start R= Fb_Axes_ItpStartStop.bBusy;
in_bAxes_ItpStartStop_Stop R= Fb_Axes_ItpStartStop.bBusy;
in_bAxes_ItpStartStop_Busy := Fb_Axes_ItpStartStop.bBusy;

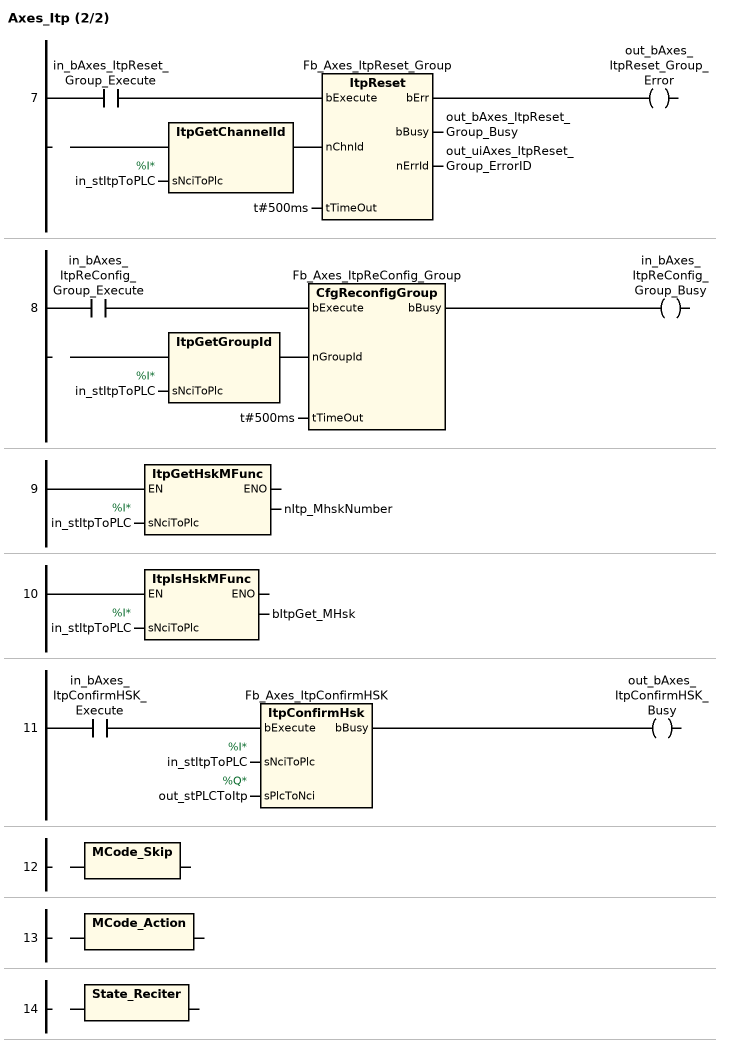
// NETWORK 7
//   in_stItpToPLC: AT %I*
Fb_Axes_ItpReset_Group(
    bExecute := in_bAxes_ItpReset_Group_Execute,
    nChnId := ItpGetChannelId(sNciToPlc := in_stItpToPLC),
    tTimeOut := t#500ms,
    bBusy => out_bAxes_ItpReset_Group_Busy,
    nErrId => out_uiAxes_ItpReset_Group_ErrorID); // ItpReset
out_bAxes_ItpReset_Group_Error := Fb_Axes_ItpReset_Group.bErr;

// NETWORK 8
//   in_stItpToPLC: AT %I*
Fb_Axes_ItpReConfig_Group(
    bExecute := in_bAxes_ItpReConfig_Group_Execute,
    nGroupId := ItpGetGroupId(sNciToPlc := in_stItpToPLC),
    tTimeOut := t#500ms); // CfgReconfigGroup
in_bAxes_ItpReConfig_Group_Busy := Fb_Axes_ItpReConfig_Group.bBusy;

// NETWORK 9
//   in_stItpToPLC: AT %I*
nItp_MhskNumber := ItpGetHskMFunc(sNciToPlc := in_stItpToPLC);

// NETWORK 10
//   in_stItpToPLC: AT %I*
bItpGet_MHsk := ItpIsHskMFunc(sNciToPlc := in_stItpToPLC);

// NETWORK 11
//   in_stItpToPLC: AT %I*
//   out_stPLCToItp: AT %Q*
Fb_Axes_ItpConfirmHSK(
    bExecute := in_bAxes_ItpConfirmHSK_Execute,
    sNciToPlc := in_stItpToPLC,
    sPlcToNci := out_stPLCToItp); // ItpConfirmHsk
out_bAxes_ItpConfirmHSK_Busy := Fb_Axes_ItpConfirmHSK.bBusy;

// NETWORK 12
MCode_Skip();

// NETWORK 13
MCode_Action();

// NETWORK 14
State_Reciter();

ACTION MCode_Action:
IF out_uiItp_Mcodenumber = 3 THEN
	out_bTOOL_HW:= TRUE;
	Axes_Itp.MCode_Skip();
END_IF

IF out_uiItp_Mcodenumber = 4 THEN
	out_bTOOL_HW:= FALSE;
	Axes_Itp.MCode_Skip();
END_IF
END_ACTION

ACTION MCode_Skip:
CASE nstep OF
	0:
		in_bAxes_ItpConfirmHSK_Execute:=FALSE;
			IF  bItpGet_MHsk AND nItp_MhskNumber =3 THEN
				nStep:=3;	
			ELSIF  bItpGet_MHsk AND nItp_MhskNumber =4 THEN
				nStep:=4;
			END_IF
	3:
		
		in_bAxes_ItpConfirmHSK_Execute:=TRUE;
			IF in_bAxes_ItpConfirmHSK_Execute AND NOT bItpGet_MHsk THEN
				nStep:=0;
			END_IF
	
	4:
		out_bTOOL_HW:= FALSE;
		in_bAxes_ItpConfirmHSK_Execute:=TRUE;
			IF in_bAxes_ItpConfirmHSK_Execute AND NOT bItpGet_MHsk THEN
				nStep:=0;
			END_IF
			
END_CASE
END_ACTION

ACTION State_Reciter:
CASE out_uiItp_InterpreterState OF
	0: out_stItp_InterpreterState_String:= "Init failed";
    1: out_stItp_InterpreterState_String:= "Idle";
    2: out_stItp_InterpreterState_String:= "Ready";
    3: out_stItp_InterpreterState_String:= "Started";
    4: out_stItp_InterpreterState_String:= "Scanning";
    5: out_stItp_InterpreterState_String:= "Running";
    6: out_stItp_InterpreterState_String:= "Stay running";
    7: out_stItp_InterpreterState_String:= "Write table";
    8: out_stItp_InterpreterState_String:= "Search line";
    9: out_stItp_InterpreterState_String:= "End";
    10:out_stItp_InterpreterState_String:= "Single Step";
    11:out_stItp_InterpreterState_String:= "Aborting";
    12:out_stItp_InterpreterState_String:= "Aborted";
    13:out_stItp_InterpreterState_String:= "Fault";
    14:out_stItp_InterpreterState_String:= "Reset";
    15:out_stItp_InterpreterState_String:= "Stop";
    16:out_stItp_InterpreterState_String:= "Wait function";
    17:out_stItp_InterpreterState_String:= "Flush buffers";
END_CASE;

IF out_wdItp_InterpolationMode=0000 THEN
	out_wdItp_InterpolationMode_string:= "Default";
    ELSIF out_wdItp_InterpolationMode=0001 THEN
    out_wdItp_InterpolationMode_string:= "SBM NC Kernel (SAF)";
    ELSIF out_wdItp_InterpolationMode=4000 THEN
    out_wdItp_InterpolationMode_string:= "SBM Block Mode Interpreter";
END_IF
END_ACTION

END_PROGRAM

// ---- POUs/Coordinate_System.TcPOU
PROGRAM Coordinate_System
VAR

END_VAR

// NETWORK 1

// NETWORK 2

END_PROGRAM

// ---- POUs/Collision_Detection.TcPOU
PROGRAM Collision_Detection
VAR
END_VAR

// NETWORK 1

ACTION High_Sensitivity:
// NETWORK 1
END_ACTION

END_PROGRAM

// ---- POUs/SoftFloat.TcPOU
PROGRAM SoftFloat
VAR
END_VAR

// NETWORK 1

END_PROGRAM

// ---- POUs/UserFrames.TcPOU
PROGRAM UserFrames
VAR
END_VAR

// NETWORK 1

END_PROGRAM

// ---- GlobalTextList.TcGTLO
TEXTLIST GlobalTextList
  58 = '      Home'
  57 = '    Home'
  59 = '  Home'
  1 = '%0.2f mm'
  17 = '%0.2f °'
  18 = '%0.3f mm'
  36 = '%d '
  34 = '%s'
  0 = '0.2f mm'
  2 = '00'
  3 = '100'
  51 = 'At Position:'
  7 = 'AuxiliaryX:'
  8 = 'AuxiliaryY:'
  9 = 'AuxiliaryZ:'
  26 = 'Build Group:'
  53 = 'Close'
  22 = 'Current Axis Position Øx:'
  23 = 'Current Axis Position Øy:'
  24 = 'Current Axis Position Øz:'
  41 = 'Current Line Number :'
  42 = 'Current MCode :'
  19 = 'Current Tool Position X:'
  20 = 'Current Tool Position Y:'
  21 = 'Current Tool Position Z:'
  38 = 'Error :'
  43 = 'Error Encountered :'
  52 = 'Execute'
  56 = 'Home'
  29 = 'Interpolation Channel:'
  40 = 'Interpolation Mode :'
  28 = 'Kinematics Channel:'
  30 = 'Load PRG:'
  4 = 'MachineX:'
  5 = 'MachineY:'
  6 = 'MachineZ:'
  10 = 'MasterAxes Enable:'
  11 = 'MasterAxes Override %:'
  45 = 'MCS Motor Access'
  44 = 'Path Velocity :'
  35 = 'Please Enter the .nc file Path Here'
  50 = 'Position Available:'
  39 = 'Present Interpreter State :'
  33 = 'Programme Name:'
  27 = 'Purge Group:'
  55 = 'Reset'
  46 = 'Reset Axes :'
  47 = 'Set X :'
  48 = 'Set Y :'
  49 = 'Set Z :'
  54 = 'Singularity Reached !'
  31 = 'Start PRG:'
  32 = 'Stop PRG:'
  37 = 'Tool Toggle:'
  12 = 'Tool X JOG +'
  15 = 'Tool X JOG -'
  13 = 'Tool Y JOG +'
  16 = 'Tool Y JOG -'
  14 = 'Tool Z JOG +'
  25 = 'Tool Z JOG -'
END_TEXTLIST

// ---- VISUs/CtrlPANEL.TcVIS
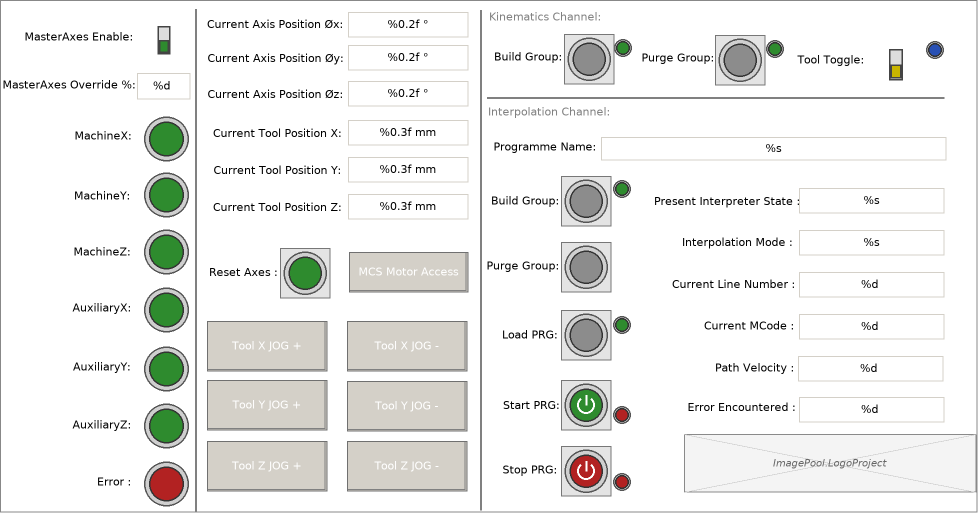
VISUALIZATION CtrlPANEL  // 978x513
    Lamp1 (137,113 59x52), variable: out_bMachX_Status, style: Lamp-Lamp1-Green
    Lamp1 (137,226 59x52), variable: out_bMachZ_Status, style: Lamp-Lamp1-Green
    Lamp1 (137,169 59x52), variable: out_bMachY_Status, style: Lamp-Lamp1-Green
    Lamp1 (137,284 59x52), variable: out_bSimsX_Status, style: Lamp-Lamp1-Green
    Lamp1 (137,343 59x52), variable: out_bSimsY_Status, style: Lamp-Lamp1-Green
    Lamp1 (137,400 59x52), variable: out_bSimsZ_Status, style: Lamp-Lamp1-Green
    DipSwitch (134,26 60x28), variable: in_bMasterAxes_Enable, behaviour: TOGGLE, style: Switch-DipSwitch-Green
    Line (196,511) (196,9)
    Label (65,121 76x30), "MachineX:"
    Label (64,181 76x30), "MachineY:"
    Label (64,237 76x30), "MachineZ:"
    Label (64,293 76x30), "AuxiliaryX:"
    Label (64,352 76x30), "AuxiliaryY:"
    Label (64,410 76x30), "AuxiliaryZ:"
    Label (19,22 120x30), "MasterAxes Enable:"
    Label (4,70 130x30), "MasterAxes Override %:"
    Button (207,321 120x50), "Tool X JOG +"
        tap in_bAxes_SimsX_Jog_Forward
    Button (207,380 120x50), "Tool Y JOG +"
        tap in_bAxes_SimsY_Jog_Forward
    Button (207,441 120x50), "Tool Z JOG +"
        tap in_bAxes_SimsZ_Jog_Forward
    Button (347,321 120x50), "Tool X JOG -"
        tap in_bAxes_SimsX_Jog_Backward
    Button (347,381 120x50), "Tool Y JOG -"
        tap in_bAxes_SimsY_Jog_Backward
    Textfield (348,12 120x25), "%0.2f °", text variable: MachX.NcToPlc.ActPos
    Textfield (348,45 120x25), "%0.2f °", text variable: MachY.NcToPlc.ActPos
    Textfield (348,81 120x25), "%0.2f °", text variable: MachZ.NcToPlc.ActPos
    Textfield (348,120 120x25), "%0.3f mm", text variable: SimsX.NcToPlc.ActPos
    Textfield (348,157 120x25), "%0.3f mm", text variable: SimsY.NcToPlc.ActPos
    Textfield (348,194 120x25), "%0.3f mm", text variable: SimsZ.NcToPlc.ActPos
    Label (211,119 133x29), "Current Tool Position X:"
    Label (211,156 133x29), "Current Tool Position Y:"
    Label (211,193 133x29), "Current Tool Position Z:"
    Label (205,10 140x29), "Current Axis Position Øx:"
    Label (209,44 133x29), "Current Axis Position Øy:"
    Label (209,80 133x29), "Current Axis Position Øz:"
    Line (481,510) (481,10)
    Button (347,441 120x50), "Tool Z JOG -"
        tap in_bAxes_SimsZ_Jog_Backward
    Label (460,42 136x30), "Build Group:"
    Lamp1 (613,38 20x20), variable: out_bAxes_KinConfigGroup_Done_HMI, style: Lamp-Lamp1-Green
    Label (619,41 118x34), "Purge Group:"
    PushSwitch (715,35 50x50), variable: in_bAxes_KinResetGroup_Execute, behaviour: TAP, style: Switch-PushSwitch-Gray
    Lamp1 (765,39 20x20), variable: out_bAxes_KinResetGroup_Done, style: Lamp-Lamp1-Green
    Line (944,98) (487,98)
    Label (477,2 136x30), "Kinematics Channel:"
    Label (481,97 136x30), "Interpolation Channel:"
    PushSwitch (561,310 50x50), variable: in_bAxes_ItpLoadPRG_Execute, behaviour: TOGGLE, style: Switch-PushSwitch-Gray
    Lamp1 (612,405 20x20), variable: in_bAxes_ItpStartStop_Error, style: Lamp-Lamp1-Red
    Label (457,186 136x30), "Build Group:"
    Label (462,320 136x30), "Load PRG:"
    Label (464,390 135x31), "Start PRG:"
    Label (462,455 136x30), "Stop PRG:"
    Lamp1 (612,472 20x20), variable: in_bAxes_ItpStartStop_Error, style: Lamp-Lamp1-Red
    Label (477,132 136x30), "Programme Name:"
    Textfield (601,137 345x23), "%s", tooltip "Please Enter the .nc file Path Here", text variable: in_strAxes_ItpLoadPRG_PRGPath
        OnMouseClick: write in_strAxes_ItpLoadPRG_PRGPath via VisuDialogs.Keypad
    Textfield (137,73 53x26), "%d", text variable: in_uiMasterAxes_Override
        OnMouseClick: write the text variable via VisuDialogs.Numpad
    Lamp1 (612,179 20x20), variable: out_bAxes_BuildItpGoup_Done, style: Lamp-Lamp1-Green
    DipSwitch (866,49 60x31), variable: in_bTOOL, behaviour: TOGGLE, style: Switch-DipSwitch-Yellow
    Lamp1 (925,40 20x20), variable: out_bTOOL_HW, style: Lamp-Lamp1-Blue
    Label (763,45 136x30), "Tool Toggle:"
    Lamp1 (137,458 59x52), variable: out_bAxes_Master_Error, style: Lamp-Lamp1-Red
    Label (76,467 76x30), "Error :"
    Textfield (799,188 145x25), "%s", text variable: out_stItp_InterpreterState_String
    Label (657,187 140x29), "Present Interpreter State :"
    Textfield (799,230 145x25), "%s", text variable: out_wdItp_InterpolationMode_string
    Label (667,228 141x29), "Interpolation Mode :"
    Textfield (799,272 145x25), "%d", text variable: out_uiItp_Linenumber
    Label (669,270 129x29), "Current Line Number :"
    Textfield (799,314 145x25), "%d", text variable: out_uiItp_Mcodenumber
    Label (702,312 94x28), "Current MCode :"
    Textfield (799,397 145x25), "%d", text variable: out_uiItp_ErrorEncountered
    Label (690,393 103x29), "Error Encountered :"
    Textfield (798,356 145x25), "%d", text variable: out_uiItp_Feedrate
    Label (708,354 93x28), "Path Velocity :"
    PushSwitch (561,242 50x50), variable: in_bAxes_ItpReConfig_Group_Execute, behaviour: TAP, style: Switch-PushSwitch-Gray
    Label (455,251 136x30), "Purge Group:"
    PushSwitch (564,34 50x50), variable: in_bAxes_KinConfigGroup_Execute, behaviour: TAP, style: Switch-PushSwitch-Gray
    PushSwitch (561,176 50x50), variable: in_bAxes_BuildItpGoup_Execute, behaviour: TOGGLE, style: Switch-PushSwitch-Gray
    PowerSwitch (561,380 50x50), variable: in_bAxes_ItpStartStop_Start, behaviour: TOGGLE, style: Switch-PowerSwitch-Green
    PowerSwitch (561,446 50x50), variable: in_bAxes_ItpStartStop_Stop, behaviour: TOGGLE, style: Switch-PowerSwitch-Red
    Lamp1 (612,315 20x20), variable: out_bAxes_ItpLoadPRG_DoneHMI, style: Lamp-Lamp1-Green
    Button (349,252 119x40), "MCS Motor Access"
        toggle in_b_MoveHome
        OnMouseClick: OpenDialog Dialog=Home, OpenModal=True, OpenCentered=True
    PushSwitch (280,248 50x50), variable: Axes_Reset_All, behaviour: TAP, style: Switch-PushSwitch-Green
    Label (192,258 103x29), "Reset Axes :"
    Image (684,434 292x58), image: ImagePool.LogoProject
END_VISUALIZATION

// ---- VISUs/Home.TcVIS
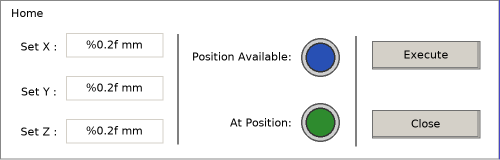
VISUALIZATION Home  // 500x160
    Rectangle (0,0 500x159)
    Label (-36,32 150x30), "Set X :"
    Label (-36,77 150x30), "Set Y :"
    Label (-36,117 150x30), "Set Z :"
    Textfield (66,33 97x24), "%0.2f mm", text variable: Set_Pos_XHome
        OnMouseDown: write Set_Pos_XHome via VisuDialogs.Numpad
    Textfield (66,76 97x24), "%0.2f mm", text variable: Set_Pos_YHome
        OnMouseClick: write Set_Pos_YHome via VisuDialogs.Numpad
    Textfield (66,119 97x24), "%0.2f mm", text variable: Set_Pos_ZHome
        OnMouseClick: write Set_Pos_ZHome via VisuDialogs.Numpad
    Line (192,47)
    Line (178,144) (178,34)
    Lamp1 (298,35 45x45), variable: Home.Pos_Exists, style: Lamp-Lamp1-Blue
    Label (167,42 150x30), "Position Available:"
    Line (192,109)
    Lamp1 (298,100 45x45), variable: out_b_inHome, style: Lamp-Lamp1-Green
    Label (206,107 110x32), "At Position:"
    Line (356,146) (356,36)
    Button (372,41 108x28), "Execute", invisible if: Home.Pos_NotValid
        toggle in_b_MoveHome
    Button (372,110 108x28), "Close"
        OnMouseClick: CloseDialog Dialog=Home, Result=OK, NumpadKeypadSet=True
    Rectangle (1,1 498x25), "Home"
END_VISUALIZATION
